FUNCTION TryConvert_DWORD_TO_BOOL : BOOL
VAR_INPUT
	in : DWORD;
	out : REFERENCE TO BOOL;
END_VAR

out := DWORD_TO_BOOL(in);
TryConvert_DWORD_TO_BOOL := TRUE;

END_FUNCTION

(* stored: Version 1.1.0.1, ProductVersion 3.1.4024.12
   POU TryConvert_DWORD_TO_BOOL: Id {aab910c7-4472-4bf5-8731-01ba14139c71}, SpecialFunc None *)
